TYPE "UDT_ScannerInterface"
VERSION : 0.1
   STRUCT
      Trigger { ExternalAccessible := 'False'; ExternalVisible := 'False'; ExternalWritable := 'False'} : Bool;
      BarCodeValue { ExternalAccessible := 'False'; ExternalVisible := 'False'; ExternalWritable := 'False'} : String;
   END_STRUCT;

END_TYPE

